// SIMATIC STEP 7 (V5.x) project BINARY DISTIL_ORIGINAL
// CPU: CPU 315-2 PN/DP
// station: Hardware
// station: SIMATIC 300(1)
// station: P_ADR_BUS
// program: S7 Program(1)

SYMBOL_TABLE
"BIN DISTILLATION"	FB 1	FB 1
"PRO_STP_BIT"	M 0.6	BOOL
END_SYMBOL_TABLE

FUNCTION_BLOCK "BIN DISTILLATION"	// FB 1
VERSION : 0.1
VAR_INPUT
  START : BOOL ;
  LL : BOOL ;
  LH : BOOL ;
  TL : BOOL ;
  TH : BOOL ;
END_VAR
VAR_OUTPUT
  V1_REBOILER : BOOL ;
  V2_CONDENSOR : BOOL ;
  V3_REFLUX : BOOL ;
  V4_DIST_PRODUCT : BOOL ;
  V5_BOTT_PRODUCT : BOOL ;
  V6_FEED : BOOL ;
END_VAR
BEGIN
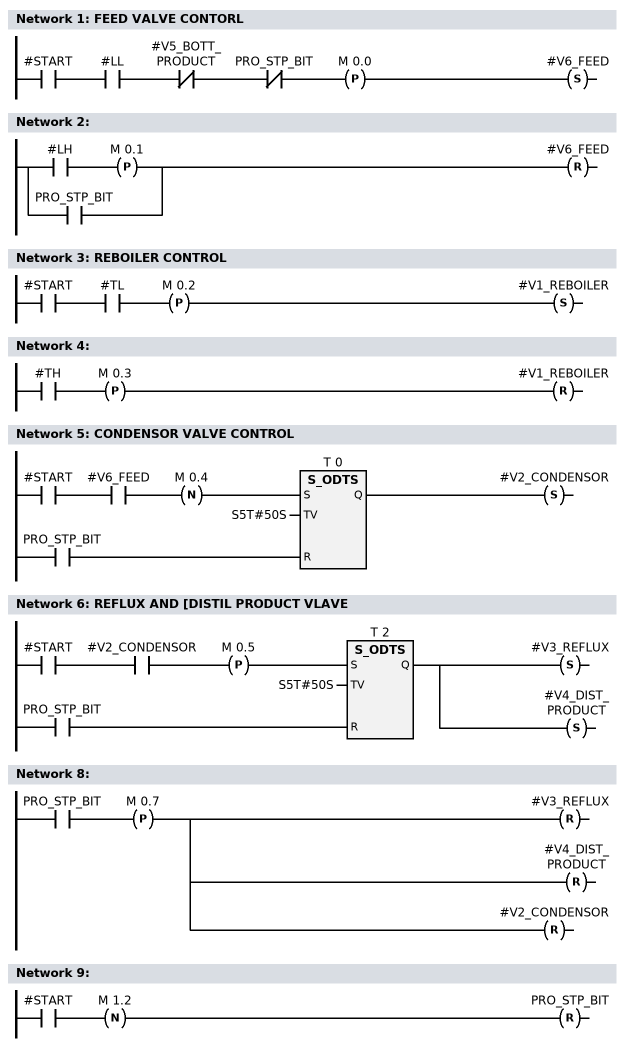
NETWORK
TITLE = FEED VALVE CONTORL
      A     #START;
      A     #LL;
      AN    #V5_BOTT_PRODUCT;
      AN    "PRO_STP_BIT";
      FP    M 0.0;
      S     #V6_FEED;
NETWORK
TITLE =
      A     #LH;
      FP    M 0.1;
      O     "PRO_STP_BIT";
      R     #V6_FEED;
NETWORK
TITLE = REBOILER CONTROL
      A     #START;
      A     #TL;
      FP    M 0.2;
      S     #V1_REBOILER;
NETWORK
TITLE =
      A     #TH;
      FP    M 0.3;
      R     #V1_REBOILER;
NETWORK
TITLE = CONDENSOR VALVE CONTROL
      A     #START;
      A     #V6_FEED;
      FN    M 0.4;
      L     S5T#50S;
      SS    T 0;
      A     "PRO_STP_BIT";
      R     T 0;
      NOP   0;
      NOP   0;
      A     T 0;
      S     #V2_CONDENSOR;
NETWORK
TITLE = REFLUX AND [DISTIL PRODUCT VLAVE
      A     #START;
      A     #V2_CONDENSOR;
      FP    M 0.5;
      L     S5T#50S;
      SS    T 2;
      A     "PRO_STP_BIT";
      R     T 2;
      NOP   0;
      NOP   0;
      A     T 2;
      S     #V3_REFLUX;
      S     #V4_DIST_PRODUCT;
NETWORK
TITLE = PROCESS STOP CONTROL
      A(;
      A     #LL;
      CU    C 0;
      BLD   101;
      NOP   0;
      NOP   0;
      A     "PRO_STP_BIT";
      R     C 0;
      L     C 0;
      T     MW 10;
      NOP   0;
      A     C 0;
      );
      A(;
      L     MW 10;
      L     2;
      ==I;
      );
      S     "PRO_STP_BIT";
NETWORK
TITLE =
      A     "PRO_STP_BIT";
      FP    M 0.7;
      R     #V3_REFLUX;
      R     #V4_DIST_PRODUCT;
      R     #V2_CONDENSOR;
NETWORK
TITLE =
      A     #START;
      FN    M 1.2;
      R     "PRO_STP_BIT";
END_FUNCTION_BLOCK

DATA_BLOCK DB 1
VERSION : 0.0
"BIN DISTILLATION"
BEGIN
END_DATA_BLOCK

ORGANIZATION_BLOCK OB 1
TITLE = "Main Program Sweep (Cycle)"
VERSION : 0.1
VAR_TEMP
  OB1_EV_CLASS : BYTE ;	//Bits 0-3 = 1 (Coming event), Bits 4-7 = 1 (Event class 1)
  OB1_SCAN_1 : BYTE ;	//1 (Cold restart scan 1 of OB 1), 3 (Scan 2-n of OB 1)
  OB1_PRIORITY : BYTE ;	//Priority of OB Execution
  OB1_OB_NUMBR : BYTE ;	//1 (Organization block 1, OB1)
  OB1_RESERVED_1 : BYTE ;	//Reserved for system
  OB1_RESERVED_2 : BYTE ;	//Reserved for system
  OB1_PREV_CYCLE : INT ;	//Cycle time of previous OB1 scan (milliseconds)
  OB1_MIN_CYCLE : INT ;	//Minimum cycle time of OB1 (milliseconds)
  OB1_MAX_CYCLE : INT ;	//Maximum cycle time of OB1 (milliseconds)
  OB1_DATE_TIME : DATE_AND_TIME ;	//Date and time OB1 started
END_VAR
BEGIN
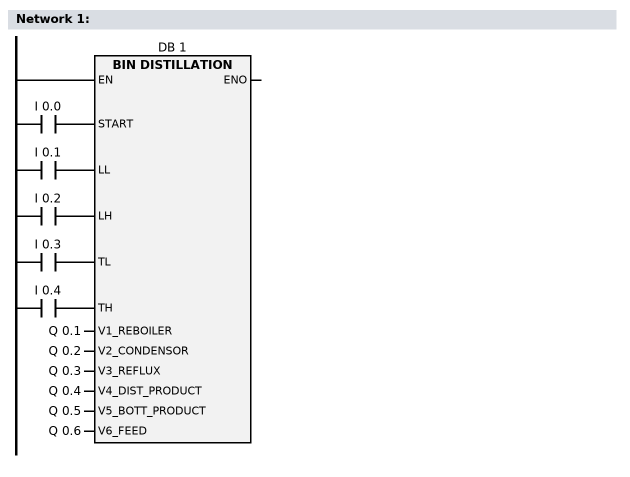
NETWORK
TITLE =
      A     I 0.0;
      =     L 20.0;
      BLD   103;
      A     I 0.1;
      =     L 20.1;
      BLD   103;
      A     I 0.2;
      =     L 20.2;
      BLD   103;
      A     I 0.3;
      =     L 20.3;
      BLD   103;
      A     I 0.4;
      =     L 20.4;
      BLD   103;
      CALL  "BIN DISTILLATION" , DB 1 (
           START                    := L 20.0,
           LL                       := L 20.1,
           LH                       := L 20.2,
           TL                       := L 20.3,
           TH                       := L 20.4,
           V1_REBOILER              := Q 0.1,
           V2_CONDENSOR             := Q 0.2,
           V3_REFLUX                := Q 0.3,
           V4_DIST_PRODUCT          := Q 0.4,
           V5_BOTT_PRODUCT          := Q 0.5,
           V6_FEED                  := Q 0.6);
      NOP   0;
END_ORGANIZATION_BLOCK
